{attribute 'linkalways'} 
{attribute 'no_explicit_call' := 'This FB is a CLASS and must be accessed using methods or properties'}
{attribute 'enable_dynamic_creation'}
FUNCTION_BLOCK DatatypeNodeFactory IMPLEMENTS I_EventHandler
VAR
	datatypes : I_Datatypes;
	nodeFactory : I_NodeFactory;
	selfCreatedNodes : Stack;
END_VAR

METHOD PROTECTED CreateAliasArrayBundleNode : I_Node
VAR_INPUT
	NodeDatatype : I_AliasDatatype;
END_VAR
VAR
	pAnyBundleNode : POINTER TO AnyAliasArrayBundleNode;
END_VAR
pAnyBundleNode := __NEW(AnyAliasArrayBundleNode(AliasDatatype := NodeDatatype));
CreateAliasArrayBundleNode := pAnyBundleNode^;
END_METHOD

METHOD PROTECTED CreateAliasArrayUnbundleNode : I_Node
VAR_INPUT
	NodeDatatype : I_AliasDatatype;
END_VAR
VAR
	pAnyUnbundleNode : POINTER TO AnyAliasArrayUnbundleNode;
END_VAR
pAnyUnbundleNode := __NEW(AnyAliasArrayUnbundleNode(AliasDatatype := NodeDatatype));
CreateAliasArrayUnbundleNode := pAnyUnbundleNode^;
END_METHOD

METHOD PROTECTED CreateAliasStructureBundleNode : I_Node
VAR_INPUT
	NodeDatatype : I_AliasDatatype;
END_VAR
VAR
	pAnyBundleNode : POINTER TO AnyAliasStructureBundleNode;
END_VAR
pAnyBundleNode := __NEW(AnyAliasStructureBundleNode(AliasDatatype := NodeDatatype));
CreateAliasStructureBundleNode := pAnyBundleNode^;
END_METHOD

METHOD PROTECTED CreateAliasStructureUnbundleNode : I_Node
VAR_INPUT
	NodeDatatype : I_AliasDatatype;
END_VAR
VAR
	pAnyUnbundleNode : POINTER TO AnyAliasStructureUnbundleNode;
END_VAR
pAnyUnbundleNode := __NEW(AnyAliasStructureUnbundleNode(AliasDatatype := NodeDatatype));
CreateAliasStructureUnbundleNode := pAnyUnbundleNode^;
END_METHOD

METHOD PROTECTED CreateArrayBundleNode : I_Node
VAR_INPUT
	NodeDatatype : I_ArrayDatatype;
END_VAR
VAR
	pAnyBundleNode : POINTER TO AnyArrayBundleNode;
END_VAR
pAnyBundleNode := __NEW(AnyArrayBundleNode(ArrayDatatype := NodeDatatype));
CreateArrayBundleNode := pAnyBundleNode^;
END_METHOD

METHOD PROTECTED CreateArrayUnbundleNode : I_Node
VAR_INPUT
	NodeDatatype : I_ArrayDatatype;
END_VAR
VAR
	pAnyUnbundleNode : POINTER TO AnyArrayUnbundleNode;
END_VAR
pAnyUnbundleNode := __NEW(AnyArrayUnbundleNode(ArrayDatatype := NodeDatatype));
CreateArrayUnbundleNode := pAnyUnbundleNode^;
END_METHOD

METHOD PROTECTED CreateDisplayNode : I_Node
VAR_INPUT
	NodeDatatype : I_Datatype;
END_VAR
VAR
	pAnyDisplayNode : POINTER TO AnyDisplayNode;
END_VAR
pAnyDisplayNode := __NEW(AnyDisplayNode(Datatype := NodeDatatype));
CreateDisplayNode := pAnyDisplayNode^;
END_METHOD

METHOD PROTECTED CreateInterfaceDisplayNode : I_Node
VAR_INPUT
	NodeDatatype : I_InterfaceDatatype;
END_VAR
VAR
	pAnyInterfaceDisplayNode : POINTER TO AnyInterfaceDisplayNode;
END_VAR
pAnyInterfaceDisplayNode := __NEW(AnyInterfaceDisplayNode(Datatype := NodeDatatype));
CreateInterfaceDisplayNode := pAnyInterfaceDisplayNode^;
END_METHOD

METHOD PROTECTED CreateLiteralNode : I_Node
VAR_INPUT
	NodeDatatype : I_Datatype;
END_VAR
VAR
	pAnyLiteralNode : POINTER TO AnyLiteralNode;
END_VAR
pAnyLiteralNode := __NEW(AnyLiteralNode(Datatype := NodeDatatype));
CreateLiteralNode := pAnyLiteralNode^;
END_METHOD

METHOD PROTECTED CreateStructureBundleNode : I_Node
VAR_INPUT
	NodeDatatype : I_StructuredDatatype;
END_VAR
VAR
	pAnyBundleNode : POINTER TO AnyStructureBundleNode;
END_VAR
pAnyBundleNode := __NEW(AnyStructureBundleNode(StructuredDatatype := NodeDatatype));
CreateStructureBundleNode := pAnyBundleNode^;
END_METHOD

METHOD PROTECTED CreateStructureUnbundleNode : I_Node
VAR_INPUT
	NodeDatatype : I_StructuredDatatype;
END_VAR
VAR
	pAnyUnbundleNode : POINTER TO AnyStructureUnbundleNode;
END_VAR
pAnyUnbundleNode := __NEW(AnyStructureUnbundleNode(StructuredDatatype := NodeDatatype));
CreateStructureUnbundleNode := pAnyUnbundleNode^;
END_METHOD

METHOD PRIVATE DeregisterWithDatatypes
VAR_INPUT
END_VAR
IF datatypes = 0 THEN
	RETURN;
END_IF

datatypes.OffEvent('OnDatatypeAdded', THIS^);
datatypes := 0;
END_METHOD

METHOD PRIVATE DisposeSelfCreatedNodes : BOOL
VAR
	node : I_Node;
END_VAR
WHILE selfCreatedNodes.TryPop(node) DO
	node.Dispose();
END_WHILE
END_METHOD

METHOD FB_exit : BOOL
VAR_INPUT
	bInCopyCode : BOOL; // if TRUE, the exit method is called for exiting an instance that is copied afterwards (online change).
END_VAR
IF bInCopyCode THEN
	RETURN;
END_IF

DeregisterWithDatatypes();
DisposeSelfCreatedNodes();
END_METHOD

METHOD FB_init : BOOL
VAR_INPUT
	bInitRetains : BOOL; // if TRUE, the retain variables are initialized (warm start / cold start)
	bInCopyCode : BOOL;  // if TRUE, the instance afterwards gets moved into the copy code (online change)
	Datatypes : I_Datatypes;
	NodeFactory : I_NodeFactory;	
END_VAR
THIS^.datatypes := Datatypes;
THIS^.nodeFactory := NodeFactory;

RegisterWithDatatypes();
END_METHOD

METHOD PUBLIC HandleEvent
VAR_INPUT
	Event : I_Event;
END_VAR
VAR
	datatypeAddedEvent : I_DatatypeAddedEvent;
	primitiveDatatype : I_Datatype;
	aliasDatatypeAddedEvent : I_AliasDatatypeAddedEvent;
	aliasDatatype : I_AliasDatatype;
	enumDatatypeAddedEvent : I_EnumDatatypeAddedEvent;
	enumDatatype : I_EnumDatatype;
	structuredDatatypeAddedEvent : I_StructuredDatatypeAddedEvent;
	structureDatatype : I_StructuredDatatype;
	interfaceDatatypeAddedEvent : I_InterfaceDatatypeAddedEvent;
	interfaceDatatype : I_InterfaceDatatype;
	arrayDatatypeAddedEvent : I_ArrayDatatypeAddedEvent;
	arrayDatatype : I_ArrayDatatype;
END_VAR
IF __QUERYINTERFACE(event, aliasDatatypeAddedEvent) THEN
	aliasDatatype := aliasDatatypeAddedEvent.Target;
	RegisterUdtLiteralNodeOfType(aliasDatatype);
	RegisterUdtDisplayNodeOfType(aliasDatatype);
	
	// at this point we have the lowest level alias who's base type is not alias (or we reached a breakout)
	IF aliasDatatype.Root.TryResolveAsArrayDatatype(arrayDatatype) THEN
		RegisterAliasArrayBundleNodeOfType(aliasDatatype);
		RegisterAliasArrayUnbundleNodeOfType(aliasDatatype);
	ELSIF aliasDatatype.Root.TryResolveAsStructuredDatatype(structureDatatype) THEN
		RegisterAliasStructureBundleNodeOfType(aliasDatatype);
		RegisterAliasStructureUnbundleNodeOfType(aliasDatatype);
	END_IF
		
	RETURN;
END_IF

IF __QUERYINTERFACE(event, enumDatatypeAddedEvent) THEN
	enumDatatype := enumDatatypeAddedEvent.Target;
	RegisterUdtLiteralNodeOfType(enumDatatype);
	RegisterUdtDisplayNodeOfType(enumDatatype);
	RETURN;
END_IF

IF __QUERYINTERFACE(event, interfaceDatatypeAddedEvent) THEN
	interfaceDatatype := interfaceDatatypeAddedEvent.Target;
	RegisterInterfaceLiteralNodeOfType(interfaceDatatype);
	RegisterInterfaceDisplayNodeOfType(interfaceDatatype);
	RETURN;
END_IF

IF __QUERYINTERFACE(event, structuredDatatypeAddedEvent) THEN
	structureDatatype := structuredDatatypeAddedEvent.Target;
	RegisterUdtLiteralNodeOfType(structureDatatype);
	RegisterUdtDisplayNodeOfType(structureDatatype);
	RegisterStructureBundleNodeOfType(structureDatatype);
	RegisterStructureUnbundleNodeOfType(structureDatatype);
	RETURN;
END_IF

IF __QUERYINTERFACE(event, arrayDatatypeAddedEvent) THEN
	RegisterUdtLiteralNodeOfType(arrayDatatypeAddedEvent.Target);
	RegisterUdtDisplayNodeOfType(arrayDatatypeAddedEvent.Target);
	RegisterArrayBundleNodeOfType(arrayDatatypeAddedEvent.Target);
	RegisterArrayUnbundleNodeOfType(arrayDatatypeAddedEvent.Target);
	RETURN;
END_IF

IF __QUERYINTERFACE(event, datatypeAddedEvent) THEN
	primitiveDatatype := datatypeAddedEvent.Target;
	RegisterPrimitiveLiteralNodeOfType(primitiveDatatype);
	RegisterPrimitiveDisplayNodeOfType(primitiveDatatype);
	RETURN;
END_IF
END_METHOD

METHOD PROTECTED RegisterAliasArrayBundleNodeOfType
VAR_INPUT
	AliasDatatype : I_AliasDatatype;
END_VAR
VAR
	node : I_Node;
	path : T_MAXSTRING;
END_VAR
node := CreateAliasArrayBundleNode(AliasDatatype);
selfCreatedNodes.Push(node);
path := concat('Bundle/', AliasDatatype.Identifier);
nodeFactory.AddNodeAsPrototype(path,node);
END_METHOD

METHOD PROTECTED RegisterAliasArrayUnbundleNodeOfType
VAR_INPUT
	AliasDatatype : I_AliasDatatype;
END_VAR
VAR
	node : I_Node;
	path : T_MAXSTRING;
END_VAR
node := CreateAliasArrayUnbundleNode(AliasDatatype);
selfCreatedNodes.Push(node);
path := concat('Unbundle/', AliasDatatype.Identifier);
nodeFactory.AddNodeAsPrototype(path,node);
END_METHOD

METHOD PROTECTED RegisterAliasStructureBundleNodeOfType
VAR_INPUT
	AliasDatatype : I_AliasDatatype;
END_VAR
VAR
	node : I_Node;
	path : T_MAXSTRING;
END_VAR
node := CreateAliasStructureBundleNode(AliasDatatype);
selfCreatedNodes.Push(node);
path := concat('Bundle/', AliasDatatype.Identifier);
nodeFactory.AddNodeAsPrototype(path,node);
END_METHOD

METHOD PROTECTED RegisterAliasStructureUnbundleNodeOfType
VAR_INPUT
	AliasDatatype : I_AliasDatatype;
END_VAR
VAR
	node : I_Node;
	path : T_MAXSTRING;
END_VAR
node := CreateAliasStructureUnbundleNode(AliasDatatype);
selfCreatedNodes.Push(node);
path := concat('Unbundle/', AliasDatatype.Identifier);
nodeFactory.AddNodeAsPrototype(path,node);
END_METHOD

METHOD PROTECTED RegisterArrayBundleNodeOfType
VAR_INPUT
	NodeDatatype : I_ArrayDatatype;
END_VAR
VAR
	node : I_Node;
	path : T_MAXSTRING;
END_VAR
node := CreateArrayBundleNode(NodeDatatype);
selfCreatedNodes.Push(node);
path := concat('Bundle/', NodeDatatype.Identifier);
nodeFactory.AddNodeAsPrototype(path,node);
END_METHOD

METHOD PROTECTED RegisterArrayUnbundleNodeOfType
VAR_INPUT
	NodeDatatype : I_ArrayDatatype;
END_VAR
VAR
	node : I_Node;
	path : T_MAXSTRING;
END_VAR
node := CreateArrayUnbundleNode(NodeDatatype);
selfCreatedNodes.Push(node);
path := concat('Unbundle/', NodeDatatype.Identifier);
nodeFactory.AddNodeAsPrototype(path,node);
END_METHOD

METHOD PROTECTED RegisterInterfaceDisplayNodeOfType
VAR_INPUT
	NodeDatatype : I_InterfaceDatatype;
END_VAR
VAR
	node : I_Node;
	path : T_MAXSTRING;
END_VAR
node := CreateInterfaceDisplayNode(NodeDatatype);
selfCreatedNodes.Push(node);
path := concat('Display/', NodeDatatype.Identifier);
nodeFactory.AddNodeAsPrototype(path,node);
END_METHOD

METHOD PROTECTED RegisterInterfaceLiteralNodeOfType
VAR_INPUT
	NodeDatatype : I_InterfaceDatatype;
END_VAR
VAR
	node : I_Node;
	path : T_MAXSTRING;
END_VAR
node := CreateLiteralNode(NodeDatatype);
selfCreatedNodes.Push(node);
path := concat('Literal/', NodeDatatype.Identifier);
nodeFactory.AddNodeAsPrototype(path,node);
END_METHOD

METHOD PROTECTED RegisterPrimitiveDisplayNodeOfType
VAR_INPUT
	NodeDatatype : I_Datatype;
END_VAR
VAR
	node : I_Node;
	path : T_MAXSTRING;
END_VAR
node := CreateDisplayNode(NodeDatatype);
selfCreatedNodes.Push(node);
path := concat('Display/', NodeDatatype.TypeName);
nodeFactory.AddNodeAsPrototype(path,node);
END_METHOD

METHOD PROTECTED RegisterPrimitiveLiteralNodeOfType
VAR_INPUT
	NodeDatatype : I_Datatype;
END_VAR
VAR
	node : I_Node;
	path : T_MAXSTRING;
END_VAR
node := CreateLiteralNode(NodeDatatype);
selfCreatedNodes.Push(node);
path := concat('Literal/', NodeDatatype.TypeName);
nodeFactory.AddNodeAsPrototype(path,node);
END_METHOD

METHOD PROTECTED RegisterStructureBundleNodeOfType
VAR_INPUT
	NodeDatatype : I_StructuredDatatype;
END_VAR
VAR
	node : I_Node;
	path : T_MAXSTRING;
END_VAR
node := CreateStructureBundleNode(NodeDatatype);
selfCreatedNodes.Push(node);
path := concat('Bundle/', NodeDatatype.Identifier);
nodeFactory.AddNodeAsPrototype(path,node);
END_METHOD

METHOD PROTECTED RegisterStructureUnbundleNodeOfType
VAR_INPUT
	NodeDatatype : I_StructuredDatatype;
END_VAR
VAR
	node : I_Node;
	path : T_MAXSTRING;
END_VAR
node := CreateStructureUnbundleNode(NodeDatatype);
selfCreatedNodes.Push(node);
path := concat('Unbundle/', NodeDatatype.Identifier);
nodeFactory.AddNodeAsPrototype(path,node);
END_METHOD

METHOD PROTECTED RegisterUdtDisplayNodeOfType
VAR_INPUT
	NodeDatatype : I_UserDefinedDatatype;
END_VAR
VAR
	node : I_Node;
	path : T_MAXSTRING;
END_VAR
node := CreateDisplayNode(NodeDatatype);
selfCreatedNodes.Push(node);
path := concat('Display/', NodeDatatype.Identifier);
nodeFactory.AddNodeAsPrototype(path,node);
END_METHOD

METHOD PROTECTED RegisterUdtLiteralNodeOfType
VAR_INPUT
	NodeDatatype : I_UserDefinedDatatype;
END_VAR
VAR
	node : I_Node;
	path : T_MAXSTRING;
END_VAR
node := CreateLiteralNode(NodeDatatype);
selfCreatedNodes.Push(node);
path := concat('Literal/', NodeDatatype.Identifier);
nodeFactory.AddNodeAsPrototype(path,node);
END_METHOD

METHOD PRIVATE RegisterWithDatatypes
VAR_INPUT
END_VAR
IF datatypes = 0 THEN
	RETURN;
END_IF

datatypes.OnEvent('OnDatatypeAdded', THIS^);
END_METHOD

END_FUNCTION_BLOCK

(* stored: Version 1.1.0.1, ProductVersion 3.1.4024.13
   POU DatatypeNodeFactory: Id {4b37bcb1-5b3c-084f-07b9-ae97280523f0}, SpecialFunc None
   Folder Constructor: Id {e3789508-846c-0b51-2172-792a6f0219f8}
   Folder Destructor: Id {701769ec-9c4f-0439-3c64-bffc00c04cc1}
   Folder Private: Id {4b06c450-3c9d-05a3-396d-cb8d55dbfe99}
   Folder Protected: Id {cd03c763-398a-08df-367f-955179e76b46}
   Method CreateAliasArrayBundleNode: Id {d91f6f5c-b069-022b-02b0-837695d66ec4}
   Method CreateAliasArrayUnbundleNode: Id {e707dfbd-1beb-05e8-3daa-331eb22d4a44}
   Method CreateAliasStructureBundleNode: Id {c1ec121a-fbd2-0600-2fdb-dcd07cfd88b7}
   Method CreateAliasStructureUnbundleNode: Id {40cd8a6c-73a2-05d7-05b2-7fb8614c17b8}
   Method CreateArrayBundleNode: Id {e5b29f80-1b2d-01b9-2f29-0873e73e2153}
   Method CreateArrayUnbundleNode: Id {ad556d76-f2d4-0873-2393-b46e303dfe51}
   Method CreateDisplayNode: Id {f5bc0ba5-7ab2-0bcf-066f-b58003dd2c5a}
   Method CreateInterfaceDisplayNode: Id {47793241-fb5b-0de0-300e-5cabec018061}
   Method CreateLiteralNode: Id {c52fa6c0-781b-0d47-0d80-60de41af51f8}
   Method CreateStructureBundleNode: Id {83d7bec4-800e-07e4-1251-d19d776aaebf}
   Method CreateStructureUnbundleNode: Id {8cd0562e-322b-0354-0533-ad232dd1bace}
   Method DeregisterWithDatatypes: Id {d281941f-7d1b-0268-2c8d-f7207a072f5a}
   Method DisposeSelfCreatedNodes: Id {a525719b-3852-0c1a-02d2-da99c688807e}
   Method FB_exit: Id {9d20964f-f8ef-0067-23b5-16439e649fce}
   Method FB_init: Id {82b14753-77c4-0521-20cf-034a973976ca}
   Method HandleEvent: Id {3ed2b7a8-ed88-0dfd-0753-1eb08b58ec83}
   Method RegisterAliasArrayBundleNodeOfType: Id {954de1eb-4c41-0cca-289c-865f8db6e544}
   Method RegisterAliasArrayUnbundleNodeOfType: Id {46101f08-133c-03e0-024c-4aa329164013}
   Method RegisterAliasStructureBundleNodeOfType: Id {78fd56dc-3ec7-0403-2845-c9223880cd60}
   Method RegisterAliasStructureUnbundleNodeOfType: Id {7915d208-88b8-097f-3ff7-7eee6f424cd1}
   Method RegisterArrayBundleNodeOfType: Id {e449e57b-91e6-0b1f-114b-7384f6362ffc}
   Method RegisterArrayUnbundleNodeOfType: Id {2d68de51-073f-0ab9-069d-f8bab82ee4d2}
   Method RegisterInterfaceDisplayNodeOfType: Id {7be2175b-0a3b-02e2-1c61-137313917382}
   Method RegisterInterfaceLiteralNodeOfType: Id {56adc14e-1ed1-0ff7-38cf-3244c05df985}
   Method RegisterPrimitiveDisplayNodeOfType: Id {87ceec21-b9ce-007c-065c-0e277e7a5dd8}
   Method RegisterPrimitiveLiteralNodeOfType: Id {dda91e61-4003-0e96-067e-8b75dd3a9867}
   Method RegisterStructureBundleNodeOfType: Id {c76eb81e-9bd3-0a25-0dc6-7837d54205c1}
   Method RegisterStructureUnbundleNodeOfType: Id {473b20bb-d3d6-0876-14f0-3d4dd1a1b689}
   Method RegisterUdtDisplayNodeOfType: Id {88226159-8e0c-06ab-09a6-1ed46c9f31a9}
   Method RegisterUdtLiteralNodeOfType: Id {065152af-1dfe-001f-0f3f-26f0fa875b3a}
   Method RegisterWithDatatypes: Id {d67b5db8-9b52-0eb6-3579-8cacdc723474} *)
